FUNCTION ValueOutOfRange : BOOL
VAR_INPUT
	r_var				:REAL;
	r_Min				:REAL;
	r_Max				:REAL;
END_VAR

IF r_var >= r_Min AND r_var <= r_Max THEN
	ValueOutOfRange := FALSE;
ELSE
	ValueOutOfRange := TRUE;
END_IF

END_FUNCTION

(* stored: Version 1.1.0.1, ProductVersion 3.1.4026.18
   POU ValueOutOfRange: Id {688bf985-97e7-4389-8950-0fa55a80e377}, SpecialFunc None *)
